FUNCTION F_SetStateParams : BOOL;
VAR_INPUT
	nStateRef	:	UDINT;
	rPosition	:	REAL;
	rTolerance: REAL;
	stBeamParams	:	ST_BeamParams;
END_VAR
VAR_IN_OUT
	Table	:	FB_LinearDeviceStateTable;
END_VAR
VAR
	stDeviceState	:	ST_DeviceState;
	
END_VAR

stDeviceState.nStateRef := nStateRef;
stDeviceState.rPosition := rPosition;
stDeviceState.rTolerance := rTolerance;
stDeviceState.stReqBeamParam := stBeamParams;

Table.A_Add(
	key := nStateRef,
	putValue := stDeviceState
);

F_SetStateParams := Table.bOk;

END_FUNCTION

(* stored: Version 1.1.0.1, ProductVersion 3.1.4024.0
   POU F_SetStateParams: Id {11c4f3b8-2db3-0013-0de5-3330469a58c0}, SpecialFunc None *)
